FUNCTION_BLOCK INTERNAL FB_PrechargeState  IMPLEMENTS I_State
VAR
	pMachine				: POINTER TO FB_Machine; // Points to the state machine (THIS)
	fVSensors				: ARRAY [0..1] OF REAL;
END_VAR

METHOD PUBLIC Check
VAR
	fLoadVoltage			: REAL;
	fInputVoltage 			: REAL;
END_VAR
THIS^.SetMainContactors();
fVSensors := THIS^.pMachine^.VSensors;

fInputVoltage := fVSensors[0];
fLoadVoltage := fVSensors[1];

IF (fLoadVoltage > 1.1 * fInputVoltage) THEN
	(* If the load voltage is greater than 110% of the input voltage then we consider that there is a problem and the load is disconnected *)
	THIS^.pMachine^.Message := '[PRECHARGE] The load voltage is greater than 110 percent of the input voltage.$0A THE SYSTEM ENTERS DISCHARGE STATE';
	THIS^.pMachine^.SetState(THIS^.pMachine^.DischargeState); 
	
ELSIF (fLoadVoltage <= 1.1 * fInputVoltage AND fLoadVoltage >= 0.9502 * fInputVoltage) THEN
	THIS^.ResetTimer();
	THIS^.pMachine^.Message := '[PRECHARGE]The load voltage is within the boundaries.$0A WAITING FOR USER ACKNOWLEDGMENT TO ENTER CHARGE STATE.';
END_IF;
END_METHOD

PROPERTY PUBLIC Description : STRING
GET
Description := 'PRE-CHARGE';
END_GET
END_PROPERTY

METHOD PUBLIC FB_init
VAR_INPUT
	bInitRetains : BOOL; // if TRUE, the retain variables are initialized (warm start / cold start)
	bInCopyCode : BOOL;  // if TRUE, the instance afterwards gets moved into the copy code (online change)
	pMachine		: POINTER TO FB_Machine; // Points to the state machine (THIS)
END_VAR
THIS^.pMachine := pMachine;
END_METHOD

METHOD PUBLIC PressButton
VAR
	fLoadVoltage			: REAL;
	fInputVoltage 			: REAL;
END_VAR
fVSensors := THIS^.pMachine^.VSensors;
fInputVoltage := fVSensors[0];
fLoadVoltage := fVSensors[1];

IF (fLoadVoltage <= 1.1 * fInputVoltage AND fLoadVoltage >= 0.9502 * fInputVoltage) THEN
	THIS^.ResetTimer(); // Not necessary, here for redundancy 
	THIS^.pMachine^.SetState(THIS^.pMachine^.ChargedState);	
	THIS^.pMachine^.Message := '[PRECHARGE] Acknowledge button has been pressed. $0A SYSTEM ENTERS CHARGED STATE.';
END_IF
END_METHOD

METHOD PUBLIC PressDischarge
THIS^.pMachine^.Message := '[PRECHARGE] Discharge button has been pressed. $0A SYSTEM ENTERS DISCHARGE STATE.';
THIS^.pMachine^.SetState(THIS^.pMachine^.DischargeState);
END_METHOD

METHOD PUBLIC Reset
THIS^.pMachine^.Message := '[PRECHARGE] Reset button has been pressed. $0A SYSTEM ENTERS DISCHARGE STATE.';
THIS^.pMachine^.SetState(THIS^.pMachine^.DischargeState);
END_METHOD

METHOD PUBLIC ResetMainContactors
VAR
	nIdx				: INT;
	bMainContactors		: ARRAY[0..1] OF BOOL;
END_VAR
FOR nIdx := 0 TO 1 DO
	bMainContactors[nIdx] := FALSE; 
END_FOR

THIS^.pMachine^.MainContactors := bMainContactors;
END_METHOD

METHOD PUBLIC ResetTimer
THIS^.pMachine^.charge_TON.IN := FALSE;
END_METHOD

METHOD PUBLIC SetMainContactors
VAR
	nIdx				: INT;
	bMainContactors		: ARRAY[0..1] OF BOOL;
END_VAR
FOR nIdx := 0 TO 1 DO
	bMainContactors[nIdx] := TRUE; 
END_FOR

THIS^.pMachine^.MainContactors := bMainContactors;
END_METHOD

METHOD PUBLIC Stop
THIS^.pMachine^.SetState(THIS^.pMachine^.ErrorState);
END_METHOD

METHOD PUBLIC TimerDone
THIS^.pMachine^.Message := '[PRECHARGE] The charging time has exceeded the set limit.$0A THE SYSTEM ENTERS DISCHARGE STATE'; 		 

THIS^.ResetTimer(); 

THIS^.pMachine^.SetState(THIS^.pMachine^.DischargeState);
END_METHOD

END_FUNCTION_BLOCK

(* stored: Version 1.1.0.1, ProductVersion 3.1.4024.12
   POU FB_PrechargeState: Id {d1ebba1d-4b62-4da0-ae46-989c293d5de3}, SpecialFunc None
   Method Check: Id {fd9b2df2-42c3-40db-96cb-3b025d8e7991}
   Property Description: Id {30c72e8b-1fbc-4524-8441-614f0ae2c91e}
   Get Get: Id {98c05ff7-dc64-4257-8237-00615927e6fa}
   Method FB_init: Id {cc325abb-4390-4cef-a637-c2f3b34ae42e}
   Method PressButton: Id {8b368998-1630-4119-b689-7c30c901f5a4}
   Method PressDischarge: Id {b923a2fd-33dc-4374-b0d1-692a68123e5b}
   Method Reset: Id {4f6e847f-ae68-4fe7-afbd-3e4eaffb6f34}
   Method ResetMainContactors: Id {3e946144-0152-4ef0-b2fb-b25e3a1eb34b}
   Method ResetTimer: Id {b3bca30e-980b-4cf7-afed-1d180c2263a2}
   Method SetMainContactors: Id {c55e4912-c420-4f87-8d31-e610ee5e0fe3}
   Method Stop: Id {7563b819-8f80-4a9d-a762-cb58f7db3cfc}
   Method TimerDone: Id {d69bb403-5ea5-4558-8409-a36e124b0824} *)
